KUKA KRL data list: ps_geo_c1.dat

&ACCESS RVO1
&REL 131
&COMMENT Solda GUN C1 geometria
&PARAM DISKPATH = KRC:\R1\Program
DEFDAT  ps_geo_c1
;FOLD EXTERNAL DECLARATIONS;%{PE}%MKUKATPBASIS,%CEXT,%VCOMMON,%P
;FOLD GRIPPERTECH EXT
EXT  H50 (INT  :IN,INT  :IN,INT  :IN,GRP_TYP  :IN )
;ENDFOLD (GRIPPERTECH EXT)
;FOLD SPOTTECH EXT
EXT  USERSPOT (S_COMMAND  :IN,SPOT_TYPE  :IN )
;ENDFOLD (SPOTTECH EXT)
;FOLD BASISTECH EXT;%{PE}%MKUKATPBASIS,%CEXT,%VEXT,%P
EXT  BAS (BAS_COMMAND  :IN,REAL  :IN )
DECL INT SUCCESS
;ENDFOLD (BASISTECH EXT)
;FOLD USER EXT;%{E}%MKUKATPUSER,%CEXT,%VEXT,%P
;Make your modifications here

;ENDFOLD (USER EXT)
;ENDFOLD (EXTERNAL DECLARATIONS)

;# ============ START PATH : swp_p13050r2_l_geo_c1 =============
DECL FDAT Fswp_60_5390={TOOL_NO 2,BASE_NO 1,IPO_FRAME #BASE,POINT2[] " ",TQ_STATE FALSE}
DECL SPOT_TYPE SS_OLP1={GUN 1,PAIR #FIRST,RETR #CLO,CLO_TM 0,PGNO1 1,PRESS1 1.0,PGNO2 0,PRESS2 0.0}
DECL E6POS Xswp_60_5390={X 1793.60498,Y 1119.29797,Z -41.4300003,A -165.905701,B -75.0368805,C 75.6208725,S 6,T 51,E1 -4282.88623,E2 0.0,E3 0.0,E4 0.0,E5 0.0,E6 0.0}
DECL FDAT Fswp_60_5378={TOOL_NO 2,BASE_NO 1,IPO_FRAME #BASE,POINT2[] " "}
DECL SPOT_TYPE SS_OLP2={GUN 1,PAIR #FIRST,RETR #CLO,CLO_TM 0,PGNO1 1,PRESS1 1.0,PGNO2 0,PRESS2 0.0}
DECL E6POS Xswp_60_5378={X 1995.44397,Y 1122.11902,Z -40.4609795,A -2.36140203,B -49.9265404,C -89.8133316,S 6,T 51,E1 -4282.31592,E2 0.0,E3 0.0,E4 0.0,E5 0.0,E6 0.0}
DECL FDAT Fswp_60_5368={TOOL_NO 2,BASE_NO 1,IPO_FRAME #BASE,POINT2[] " "}
DECL SPOT_TYPE SS_OLP3={GUN 1,PAIR #FIRST,RETR #CLO,CLO_TM 0,PGNO1 1,PRESS1 1.0,PGNO2 0,PRESS2 0.0}
DECL E6POS Xswp_60_5368={X 2052.64502,Y 972.549072,Z -42.4693718,A -85.639267,B -73.5025711,C -95.7587891,S 6,T 51,E1 -4487.2959,E2 0.0,E3 0.0,E4 0.0,E5 0.0,E6 0.0}
DECL FDAT Fswp_60_5360={TOOL_NO 2,BASE_NO 1,IPO_FRAME #BASE,POINT2[] " "}
DECL SPOT_TYPE SS_OLP4={GUN 1,PAIR #FIRST,RETR #CLO,CLO_TM 0,PGNO1 1,PRESS1 1.0,PGNO2 0,PRESS2 0.0}
DECL E6POS Xswp_60_5360={X 2051.40991,Y 830.991577,Z -72.7930908,A -89.8485336,B -38.7230415,C -92.0951614,S 6,T 51,E1 -4487.2959,E2 0.0,E3 0.0,E4 0.0,E5 0.0,E6 0.0}
DECL FDAT Fswp_60_5354={TOOL_NO 2,BASE_NO 1,IPO_FRAME #BASE,POINT2[] " "}
DECL SPOT_TYPE SS_OLP5={GUN 1,PAIR #FIRST,RETR #CLO,CLO_TM 0,PGNO1 1,PRESS1 1.0,PGNO2 0,PRESS2 0.0}
DECL E6POS Xswp_60_5354={X 2052.74707,Y 687.211487,Z -69.1016464,A 89.8141937,B -4.71356201,C 90.1745834,S 6,T 51,E1 -4487.2998,E2 0.0,E3 0.0,E4 0.0,E5 0.0,E6 0.0}
DECL FDAT Fswp_60_5348={TOOL_NO 2,BASE_NO 1,IPO_FRAME #BASE,POINT2[] " "}
DECL SPOT_TYPE SS_OLP6={GUN 1,PAIR #FIRST,RETR #CLO,CLO_TM 0,PGNO1 1,PRESS1 1.0,PGNO2 0,PRESS2 0.0}
DECL E6POS Xswp_60_5348={X 2051.51196,Y 627.115173,Z -2.50994706,A 89.8144608,B -4.71358299,C 90.1741791,S 6,T 51,E1 -4487.2998,E2 0.0,E3 0.0,E4 0.0,E5 0.0,E6 0.0}
DECL FDAT Fswp_60_5342={TOOL_NO 2,BASE_NO 1,IPO_FRAME #BASE,POINT2[] " "}
DECL SPOT_TYPE SS_OLP7={GUN 1,PAIR #FIRST,RETR #CLO,CLO_TM 0,PGNO1 1,PRESS1 1.0,PGNO2 0,PRESS2 0.0}
DECL E6POS Xswp_60_5342={X 2055.79199,Y 617.443176,Z 85.3936462,A 89.999321,B -34.127739,C 90.0019379,S 6,T 51,E1 -4487.30078,E2 0.0,E3 0.0,E4 0.0,E5 0.0,E6 0.0}
DECL FDAT Fswp_60_5336={TOOL_NO 2,BASE_NO 1,IPO_FRAME #BASE,POINT2[] " "}
DECL SPOT_TYPE SS_OLP8={GUN 1,PAIR #FIRST,RETR #CLO,CLO_TM 0,PGNO1 1,PRESS1 1.0,PGNO2 0,PRESS2 0.0}
DECL E6POS Xswp_60_5336={X 2058.30298,Y 508.353699,Z 145.004395,A 89.9974213,B -46.7444382,C 90.0027695,S 6,T 51,E1 -4487.2998,E2 0.0,E3 0.0,E4 0.0,E5 0.0,E6 0.0}
DECL SPOT_TYPE SS_OLP9={GUN 1,PAIR #FIRST,RETR #CLO,CLO_TM 0,PGNO1 1,PRESS1 1.0,PGNO2 0,PRESS2 0.0}
DECL FDAT Fswp_60_5324={TOOL_NO 2,BASE_NO 1,IPO_FRAME #BASE,POINT2[] " "}
DECL SPOT_TYPE SS_OLP10={GUN 1,PAIR #FIRST,RETR #CLO,CLO_TM 0,PGNO1 1,PRESS1 1.0,PGNO2 0,PRESS2 0.0}
DECL E6POS Xswp_60_5324={X 2058.63306,Y 416.970703,Z 279.76889,A 89.9949036,B -60.1505089,C 90.006073,S 6,T 51,E1 -4487.2998,E2 0.0,E3 0.0,E4 0.0,E5 0.0,E6 0.0}
DECL FDAT Fswp_60_5318={TOOL_NO 2,BASE_NO 1,IPO_FRAME #BASE,POINT2[] " "}
DECL SPOT_TYPE SS_OLP11={GUN 1,PAIR #FIRST,RETR #CLO,CLO_TM 0,PGNO1 1,PRESS1 1.0,PGNO2 0,PRESS2 0.0}
DECL E6POS Xswp_60_5318={X 2058.04297,Y 343.247498,Z 329.933685,A -89.9762192,B -84.4996567,C -90.0254974,S 6,T 51,E1 -4487.31787,E2 0.0,E3 0.0,E4 0.0,E5 0.0,E6 0.0}
DECL FDAT Fswp_60_5312={TOOL_NO 2,BASE_NO 1,IPO_FRAME #BASE,POINT2[] " "}
DECL SPOT_TYPE SS_OLP12={GUN 1,PAIR #FIRST,RETR #CLO,CLO_TM 0,PGNO1 1,PRESS1 1.0,PGNO2 0,PRESS2 0.0}
DECL E6POS Xswp_60_5312={X 2063.91699,Y 232.038406,Z 341.721008,A -90.0093765,B -89.2421036,C -89.9965515,S 6,T 51,E1 -4487.29785,E2 0.0,E3 0.0,E4 0.0,E5 0.0,E6 0.0}
DECL BASIS_SUGG_T LAST_BASIS={POINT1[] "P0                      ",POINT2[] "P0                      ",CP_PARAMS[] "CPDAT0                  ",PTP_PARAMS[] "PDAT0                   ",CONT[] "                        ",CP_VEL[] "2.0                     ",PTP_VEL[] "100                     ",SYNC_PARAMS[] "SYNCDAT                 ",SPL_NAME[] "S0                      "}
DECL SPOT_SUGG_T LAST_SPOT={GUN[] "1                       ",RETR_CMD[] "#OPN                    ",CHOISE[] "#FIRST                  ",CLO_TM[] "1                       ",PGNO1[] "37                      ",PRESS1[] "0                       ",PGNO2[] "1                       ",PRESS2[] "0                       ",SPOT_PARAMS[] "SDAT14                  "}
DECL SPOT_TYPE SSDAT1={GUN 1,PAIR #FIRST,RETR #OPN,CLO_TM 0,PGNO1 1,PRESS1 1.0,PGNO2 0,PRESS2 0.0}
DECL SPOT_TYPE SS_OLP13={GUN 1,PAIR #FIRST,RETR #CLO,CLO_TM 0,PGNO1 1,PRESS1 1.0,PGNO2 0,PRESS2 0.0}
DECL E6POS XP6={X 14.2474098,Y -4270.53809,Z 1356.71594,A 46.7418518,B 2.44693804,C -28.1381607,S 6,T 50,E1 -2092.58911,E2 0.0,E3 0.0,E4 0.0,E5 0.0,E6 0.0}
DECL FDAT FP6={TOOL_NO 2,BASE_NO 0,IPO_FRAME #BASE,POINT2[] " ",TQ_STATE FALSE}
DECL PDAT PPDAT34={VEL 100.0,ACC 100.0,APO_DIST 10.0,APO_MODE #CDIS}
DECL E6POS XPS123={X 1975.453,Y 1262.80505,Z -89.8548737,A -7.88512707,B -42.2266693,C -81.8771667,S 6,T 51,E1 -4282.896,E2 0.0,E3 0.0,E4 0.0,E5 0.0,E6 0.0}
DECL FDAT FPS123={TOOL_NO 2,BASE_NO 1,IPO_FRAME #BASE,POINT2[] " ",TQ_STATE FALSE}
DECL PDAT PPDAT38={VEL 100.0,ACC 100.0,APO_DIST 100.0}
DECL PDAT PPDAT0={VEL 100.0,ACC 100.0,APO_DIST 100.0,APO_MODE #CDIS}
DECL E6POS XP0={X 1831.76001,Y 1986.38696,Z 157.435593,A -57.9526711,B -77.0295563,C -42.9496689,S 6,T 50,E1 -4010.88403,E2 0.0,E3 0.0,E4 0.0,E5 0.0,E6 0.0}
DECL FDAT FP0={TOOL_NO 2,BASE_NO 1,IPO_FRAME #BASE,POINT2[] " ",TQ_STATE FALSE}
DECL E6POS XP10={X 1976.64001,Y 1119.03406,Z -90.3725662,A -5.75681591,B -42.5264511,C -84.9908371,S 6,T 51,E1 -4282.896,E2 0.0,E3 0.0,E4 0.0,E5 0.0,E6 0.0}
DECL FDAT FP10={TOOL_NO 2,BASE_NO 1,IPO_FRAME #BASE,POINT2[] " ",TQ_STATE FALSE}
DECL PDAT PPDAT39={VEL 100.0,ACC 100.0,APO_DIST 50.0,APO_MODE #CDIS}
DECL PDAT PPDAT40={VEL 100.0,ACC 100.0,APO_DIST 100.0}
DECL E6POS XP11={X 1931.23596,Y 1118.84595,Z -119.764801,A -12.6583996,B -41.2317009,C -74.8182831,S 6,T 51,E1 -4282.896,E2 0.0,E3 0.0,E4 0.0,E5 0.0,E6 0.0}
DECL FDAT FP11={TOOL_NO 2,BASE_NO 1,IPO_FRAME #BASE,POINT2[] " ",TQ_STATE FALSE}
DECL PDAT PPDAT41={VEL 100.0,ACC 100.0,APO_DIST 100.0,APO_MODE #CDIS}
DECL E6POS XP12={X 1819.70203,Y 1159.33301,Z -102.061302,A -82.8152771,B -72.2565918,C -9.40070915,S 6,T 51,E1 -4282.896,E2 0.0,E3 0.0,E4 0.0,E5 0.0,E6 0.0}
DECL FDAT FP12={TOOL_NO 2,BASE_NO 1,IPO_FRAME #BASE,POINT2[] " ",TQ_STATE FALSE}
DECL PDAT PPDAT42={VEL 100.0,ACC 100.0,APO_DIST 100.0,APO_MODE #CDIS}
DECL E6POS XP13={X 1792.13,Y 1120.06299,Z -64.8214035,A -155.350403,B -74.3082733,C 64.7092438,S 6,T 51,E1 -4282.896,E2 0.0,E3 0.0,E4 0.0,E5 0.0,E6 0.0}
DECL FDAT FP13={TOOL_NO 2,BASE_NO 1,IPO_FRAME #BASE,POINT2[] " ",TQ_STATE FALSE}
DECL PDAT PPDAT43={VEL 100.0,ACC 100.0,APO_DIST 100.0,APO_MODE #CDIS}
DECL PDAT PPDAT44={VEL 100.0,ACC 100.0,APO_DIST 100.0}
DECL E6POS XP14={X 1818.04395,Y 1135.521,Z -105.700798,A -167.004501,B -43.7118111,C 71.4859467,S 6,T 51,E1 -4282.896,E2 0.0,E3 0.0,E4 0.0,E5 0.0,E6 0.0}
DECL FDAT FP14={TOOL_NO 2,BASE_NO 1,IPO_FRAME #BASE,POINT2[] " ",TQ_STATE FALSE}
DECL PDAT PPDAT45={VEL 100.0,ACC 100.0,APO_DIST 100.0,APO_MODE #CDIS}
DECL E6POS XPS000={X 1814.72803,Y 1480.03296,Z -122.856003,A -167.018295,B -43.7061081,C 71.4881973,S 6,T 50,E1 -4282.896,E2 0.0,E3 0.0,E4 0.0,E5 0.0,E6 0.0}
DECL FDAT FPS000={TOOL_NO 2,BASE_NO 1,IPO_FRAME #BASE,POINT2[] " ",TQ_STATE FALSE}
DECL PDAT PPDAT46={VEL 100.0,ACC 100.0,APO_DIST 100.0}
DECL E6POS XP15={X 2255.78809,Y 2237.59106,Z 107.454803,A -82.0964432,B -22.1816597,C -22.13521,S 6,T 50,E1 -4282.89404,E2 0.0,E3 0.0,E4 0.0,E5 0.0,E6 0.0}
DECL FDAT FP15={TOOL_NO 2,BASE_NO 1,IPO_FRAME #BASE,POINT2[] " ",TQ_STATE FALSE}
DECL PDAT PPDAT47={VEL 100.0,ACC 100.0,APO_DIST 100.0,APO_MODE #CDIS}
DECL E6POS XP16={X 3165.62207,Y 1778.36902,Z -151.722107,A 120.920898,B -1.89024901,C 8.91728306,S 6,T 51,E1 -4282.89404,E2 0.0,E3 0.0,E4 0.0,E5 0.0,E6 0.0}
DECL FDAT FP16={TOOL_NO 2,BASE_NO 1,IPO_FRAME #BASE,POINT2[] " ",TQ_STATE FALSE}
DECL PDAT PPDAT49={VEL 100.0,ACC 100.0,APO_DIST 100.0,APO_MODE #CDIS}
DECL E6POS XP17={X 2850.94189,Y 1183.13403,Z -133.184601,A 127.037201,B -29.0648193,C 14.88025,S 6,T 51,E1 -4379.94092,E2 0.0,E3 0.0,E4 0.0,E5 0.0,E6 0.0}
DECL FDAT FP17={TOOL_NO 2,BASE_NO 1,IPO_FRAME #BASE,POINT2[] " ",TQ_STATE FALSE}
DECL PDAT PPDAT50={VEL 100.0,ACC 100.0,APO_DIST 100.0,APO_MODE #CDIS}
DECL E6POS XP18={X 2507.34912,Y 900.431274,Z -270.858887,A -154.130707,B -49.1211395,C -23.3417206,S 6,T 51,E1 -4427.95215,E2 0.0,E3 0.0,E4 0.0,E5 0.0,E6 0.0}
DECL FDAT FP18={TOOL_NO 2,BASE_NO 1,IPO_FRAME #BASE,POINT2[] " ",TQ_STATE FALSE}
DECL PDAT PPDAT51={VEL 100.0,ACC 100.0,APO_DIST 100.0,APO_MODE #CDIS}
DECL E6POS XP19={X 2244.12695,Y 845.446411,Z -102.626404,A -90.2177734,B -50.6062508,C -89.3426514,S 6,T 51,E1 -4487.2998,E2 0.0,E3 0.0,E4 0.0,E5 0.0,E6 0.0}
DECL FDAT FP19={TOOL_NO 2,BASE_NO 1,IPO_FRAME #BASE,POINT2[] " ",TQ_STATE FALSE}
DECL PDAT PPDAT52={VEL 100.0,ACC 100.0,APO_DIST 100.0,APO_MODE #CDIS}
DECL E6POS XP20={X 2115.19409,Y 940.910217,Z -73.8749466,A -88.6004715,B -57.4064102,C -93.0368729,S 6,T 51,E1 -4487.29688,E2 0.0,E3 0.0,E4 0.0,E5 0.0,E6 0.0}
DECL FDAT FP20={TOOL_NO 2,BASE_NO 1,IPO_FRAME #BASE,POINT2[] " ",TQ_STATE FALSE}
DECL PDAT PPDAT53={VEL 100.0,ACC 100.0,APO_DIST 100.0,APO_MODE #CDIS}
DECL E6POS XP21={X 2047.13098,Y 942.281982,Z -76.641983,A -88.6010895,B -57.405941,C -93.0353088,S 6,T 51,E1 -4487.29688,E2 0.0,E3 0.0,E4 0.0,E5 0.0,E6 0.0}
DECL FDAT FP21={TOOL_NO 2,BASE_NO 1,IPO_FRAME #BASE,POINT2[] " ",TQ_STATE FALSE}
DECL PDAT PPDAT54={VEL 100.0,ACC 100.0,APO_DIST 100.0,APO_MODE #CDIS}
DECL E6POS XP22={X 2047.75195,Y 982.460327,Z -49.2609482,A -85.6292114,B -73.5014267,C -95.7655716,S 6,T 51,E1 -4487.29688,E2 0.0,E3 0.0,E4 0.0,E5 0.0,E6 0.0}
DECL FDAT FP22={TOOL_NO 2,BASE_NO 1,IPO_FRAME #BASE,POINT2[] " ",TQ_STATE FALSE}
DECL PDAT PPDAT55={VEL 100.0,ACC 100.0,APO_DIST 100.0,APO_MODE #CDIS}
DECL PDAT PPDAT56={VEL 100.0,ACC 100.0,APO_DIST 100.0}
DECL E6POS XP23={X 2048.30591,Y 918.138916,Z -63.4876289,A -88.6876297,B -56.5051003,C -92.9628525,S 6,T 51,E1 -4487.29688,E2 0.0,E3 0.0,E4 0.0,E5 0.0,E6 0.0}
DECL FDAT FP23={TOOL_NO 2,BASE_NO 1,IPO_FRAME #BASE,POINT2[] " ",TQ_STATE FALSE}
DECL PDAT PPDAT57={VEL 100.0,ACC 100.0,APO_DIST 100.0,APO_MODE #CDIS}
DECL E6POS XP24={X 2049.125,Y 831.437378,Z -74.7315063,A -89.8483734,B -38.7232094,C -92.0950165,S 6,T 51,E1 -4487.29688,E2 0.0,E3 0.0,E4 0.0,E5 0.0,E6 0.0}
DECL FDAT FP24={TOOL_NO 2,BASE_NO 1,IPO_FRAME #BASE,POINT2[] " ",TQ_STATE FALSE}
DECL PDAT PPDAT58={VEL 100.0,ACC 100.0,APO_DIST 20.0,APO_MODE #CDIS}
DECL PDAT PPDAT59={VEL 100.0,ACC 100.0,APO_DIST 100.0}
DECL E6POS XP25={X 2046.797,Y 858.526917,Z -100.2687,A -89.9878235,B -36.5164413,C -90.7241592,S 6,T 51,E1 -4487.29883,E2 0.0,E3 0.0,E4 0.0,E5 0.0,E6 0.0}
DECL FDAT FP25={TOOL_NO 2,BASE_NO 1,IPO_FRAME #BASE,POINT2[] " ",TQ_STATE FALSE}
DECL PDAT PPDAT60={VEL 100.0,ACC 100.0,APO_DIST 100.0,APO_MODE #CDIS}
DECL E6POS XP26={X 2159.44507,Y 857.708984,Z -101.407303,A -89.9878235,B -36.5160408,C -90.7243576,S 6,T 51,E1 -4487.29883,E2 0.0,E3 0.0,E4 0.0,E5 0.0,E6 0.0}
DECL FDAT FP26={TOOL_NO 2,BASE_NO 1,IPO_FRAME #BASE,POINT2[] " ",TQ_STATE FALSE}
DECL PDAT PPDAT61={VEL 100.0,ACC 100.0,APO_DIST 100.0,APO_MODE #CDIS}
DECL E6POS XP27={X 2146.48999,Y 788.576416,Z -75.8830719,A 89.8144608,B -4.71849298,C 90.1741867,S 6,T 51,E1 -4487.2998,E2 0.0,E3 0.0,E4 0.0,E5 0.0,E6 0.0}
DECL FDAT FP27={TOOL_NO 2,BASE_NO 1,IPO_FRAME #BASE,POINT2[] " ",TQ_STATE FALSE}
DECL PDAT PPDAT62={VEL 100.0,ACC 100.0,APO_DIST 100.0,APO_MODE #CDIS}
DECL E6POS XP28={X 2146.62695,Y 811.116272,Z -52.6086311,A -88.3386993,B -84.5875397,C -91.8407135,S 6,T 51,E1 -4487.2998,E2 0.0,E3 0.0,E4 0.0,E5 0.0,E6 0.0}
DECL FDAT FP28={TOOL_NO 2,BASE_NO 1,IPO_FRAME #BASE,POINT2[] " ",TQ_STATE FALSE}
DECL PDAT PPDAT63={VEL 100.0,ACC 100.0,APO_DIST 100.0,APO_MODE #CDIS}
DECL E6POS XP34={X 2051.16992,Y 627.691772,Z -43.1946182,A 89.8142395,B -4.71378708,C 90.1743011,S 6,T 51,E1 -4487.2998,E2 0.0,E3 0.0,E4 0.0,E5 0.0,E6 0.0}
DECL FDAT FP34={TOOL_NO 2,BASE_NO 1,IPO_FRAME #BASE,POINT2[] " ",TQ_STATE FALSE}
DECL PDAT PPDAT65={VEL 100.0,ACC 100.0,APO_DIST 100.0,APO_MODE #CDIS}
DECL PDAT PPDAT66={VEL 100.0,ACC 100.0,APO_DIST 100.0}
DECL E6POS XP35={X 2053.42993,Y 537.918091,Z 14.90874,A 89.9957962,B -33.604599,C 90.0059662,S 6,T 51,E1 -4487.2998,E2 0.0,E3 0.0,E4 0.0,E5 0.0,E6 0.0}
DECL FDAT FP35={TOOL_NO 2,BASE_NO 1,IPO_FRAME #BASE,POINT2[] " ",TQ_STATE FALSE}
DECL PDAT PPDAT67={VEL 100.0,ACC 100.0,APO_DIST 100.0,APO_MODE #CDIS}
DECL PDAT PPDAT68={VEL 100.0,ACC 100.0,APO_DIST 100.0}
DECL PDAT PPDAT69={VEL 100.0,ACC 100.0,APO_DIST 100.0}
DECL PDAT PPDAT70={VEL 100.0,ACC 100.0,APO_DIST 100.0}
DECL E6POS Xswp_60_5350={X 2057.52295,Y 450.2948,Z 220.931,A 89.9962006,B -49.0321198,C 90.0046692,S 6,T 51,E1 -4487.2998,E2 0.0,E3 0.0,E4 0.0,E5 0.0,E6 0.0}
DECL FDAT Fswp_60_5350={TOOL_NO 2,BASE_NO 1,IPO_FRAME #BASE,POINT2[] " ",TQ_STATE FALSE}
DECL E6POS XP36={X 2056.47998,Y 464.042999,Z 176.894196,A 89.9945374,B -47.4184914,C 90.0042496,S 6,T 51,E1 -4487.2998,E2 0.0,E3 0.0,E4 0.0,E5 0.0,E6 0.0}
DECL FDAT FP36={TOOL_NO 2,BASE_NO 1,IPO_FRAME #BASE,POINT2[] " ",TQ_STATE FALSE}
DECL PDAT PPDAT71={VEL 100.0,ACC 100.0,APO_DIST 100.0,APO_MODE #CDIS}
DECL PDAT PPDAT72={VEL 100.0,ACC 100.0,APO_DIST 100.0}
DECL E6POS XP37={X 2058.99902,Y 355.600891,Z 263.370087,A -89.9917908,B -84.4970779,C -90.0120468,S 6,T 51,E1 -4487.2998,E2 0.0,E3 0.0,E4 0.0,E5 0.0,E6 0.0}
DECL FDAT FP37={TOOL_NO 2,BASE_NO 1,IPO_FRAME #BASE,POINT2[] " ",TQ_STATE FALSE}
DECL PDAT PPDAT73={VEL 100.0,ACC 100.0,APO_DIST 100.0,APO_MODE #CDIS}
DECL PDAT PPDAT74={VEL 100.0,ACC 100.0,APO_DIST 100.0}
DECL E6POS XP38={X 2061.27295,Y 355.603607,Z 263.36969,A -89.986618,B -84.4975433,C -90.0177231,S 6,T 51,E1 -4487.2998,E2 0.0,E3 0.0,E4 0.0,E5 0.0,E6 0.0}
DECL FDAT FP38={TOOL_NO 2,BASE_NO 1,IPO_FRAME #BASE,POINT2[] " ",TQ_STATE FALSE}
DECL PDAT PPDAT75={VEL 100.0,ACC 100.0,APO_DIST 100.0,APO_MODE #CDIS}
DECL E6POS XP39={X 2118.13599,Y 333.994293,Z 271.6651,A 89.993927,B -68.975502,C 89.9993362,S 6,T 51,E1 -4487.29883,E2 0.0,E3 0.0,E4 0.0,E5 0.0,E6 0.0}
DECL FDAT FP39={TOOL_NO 2,BASE_NO 1,IPO_FRAME #BASE,POINT2[] " ",TQ_STATE FALSE}
DECL PDAT PPDAT76={VEL 100.0,ACC 100.0,APO_DIST 100.0,APO_MODE #CDIS}
DECL E6POS XP40={X 2075.04004,Y 270.539215,Z 300.605988,A 89.9879303,B -79.5295181,C 90.0074005,S 6,T 51,E1 -4487.29688,E2 0.0,E3 0.0,E4 0.0,E5 0.0,E6 0.0}
DECL FDAT FP40={TOOL_NO 2,BASE_NO 1,IPO_FRAME #BASE,POINT2[] " ",TQ_STATE FALSE}
DECL PDAT PPDAT77={VEL 100.0,ACC 100.0,APO_DIST 100.0,APO_MODE #CDIS}
DECL E6POS XP41={X 2059.625,Y 272.974213,Z 316.043213,A 89.9944382,B -79.5298462,C 90.000267,S 6,T 51,E1 -4487.29688,E2 0.0,E3 0.0,E4 0.0,E5 0.0,E6 0.0}
DECL FDAT FP41={TOOL_NO 2,BASE_NO 1,IPO_FRAME #BASE,POINT2[] " ",TQ_STATE FALSE}
DECL PDAT PPDAT78={VEL 100.0,ACC 100.0,APO_DIST 100.0,APO_MODE #CDIS}
DECL PDAT PPDAT79={VEL 100.0,ACC 100.0,APO_DIST 100.0}
DECL E6POS XP42={X 2063.51611,Y -5007.45508,Z 639.768799,A -73.1590881,B -24.9932995,C -19.3749294,S 6,T 51,E1 -4487.2998,E2 0.0,E3 0.0,E4 0.0,E5 0.0,E6 0.0}
DECL FDAT FP42={TOOL_NO 2,BASE_NO 0,IPO_FRAME #BASE,POINT2[] " ",TQ_STATE FALSE}
DECL PDAT PPDAT80={VEL 100.0,ACC 100.0,APO_DIST 100.0,APO_MODE #CDIS}
DECL E6POS XP43={X 2507.71899,Y -6022.83203,Z 1824.85803,A -15.74121,B -87.3473587,C -74.6977615,S 6,T 51,E1 -4487.29785,E2 0.0,E3 0.0,E4 0.0,E5 0.0,E6 0.0}
DECL FDAT FP43={TOOL_NO 2,BASE_NO 0,IPO_FRAME #BASE,POINT2[] " ",TQ_STATE FALSE}
DECL PDAT PPDAT81={VEL 100.0,ACC 100.0,APO_DIST 100.0,APO_MODE #CDIS}
DECL E6POS XP44={X 3580.86401,Y 1344.72595,Z -359.380798,A -178.304504,B 6.4053278,C -5.48929977,S 6,T 51,E1 -4064.18311,E2 0.0,E3 0.0,E4 0.0,E5 0.0,E6 0.0}
DECL FDAT FP44={TOOL_NO 2,BASE_NO 1,IPO_FRAME #BASE,POINT2[] " ",TQ_STATE FALSE}
DECL PDAT PPDAT82={VEL 100.0,ACC 100.0,APO_DIST 100.0,APO_MODE #CDIS}
DECL E6POS XP45={X 3286.89404,Y 2001.38904,Z -150.2827,A 163.915298,B -15.1394901,C 24.9498901,S 6,T 51,E1 -3093.53003,E2 0.0,E3 0.0,E4 0.0,E5 0.0,E6 0.0}
DECL FDAT FP45={TOOL_NO 2,BASE_NO 1,IPO_FRAME #BASE,POINT2[] " ",TQ_STATE FALSE}
DECL PDAT PPDAT83={VEL 100.0,ACC 100.0,APO_DIST 100.0,APO_MODE #CDIS}
DECL E6POS XP46={X -97.4183807,Y -1779.59204,Z 959.895325,A -87.2605209,B -4.11820889,C -0.3932679,S 2,T 10,E1 -303.91449,E2 0.0,E3 0.0,E4 0.0,E5 0.0,E6 0.0}
DECL FDAT FP46={TOOL_NO 2,BASE_NO 0,IPO_FRAME #BASE,POINT2[] " ",TQ_STATE FALSE}
DECL PDAT PPDAT84={VEL 100.0,ACC 100.0,APO_DIST 100.0}
DECL PDAT PPDAT86={VEL 100.0,ACC 100.0,APO_DIST 100.0,APO_MODE #CDIS}
DECL E6POS XP48={X -353.518188,Y -4054.72705,Z 1005.86902,A -168.852097,B -23.8397598,C 40.0236511,S 2,T 2,E1 -1997.07104,E2 0.0,E3 0.0,E4 0.0,E5 0.0,E6 0.0}
DECL FDAT FP48={TOOL_NO 2,BASE_NO 0,IPO_FRAME #BASE,POINT2[] " ",TQ_STATE FALSE}
DECL PDAT PPDAT87={VEL 100.0,ACC 100.0,APO_DIST 100.0}
DECL E6POS XP49={X 2050.37793,Y 688.451599,Z -119.098396,A 89.8146667,B -4.71360588,C 90.1747589,S 6,T 51,E1 -4487.29883,E2 0.0,E3 0.0,E4 0.0,E5 0.0,E6 0.0}
DECL FDAT FP49={TOOL_NO 2,BASE_NO 1,IPO_FRAME #BASE,POINT2[] " ",TQ_STATE FALSE}
DECL PDAT PPDAT88={VEL 100.0,ACC 100.0,APO_DIST 100.0,APO_MODE #CDIS}
DECL E6POS XP51={X 2332.18311,Y 353.697693,Z -173.253296,A -156.103607,B -66.3182678,C -25.5800705,S 6,T 51,E1 -4487.29883,E2 0.0,E3 0.0,E4 0.0,E5 0.0,E6 0.0}
DECL FDAT FP51={TOOL_NO 2,BASE_NO 1,IPO_FRAME #BASE,POINT2[] " ",TQ_STATE FALSE}
DECL PDAT PPDAT90={VEL 100.0,ACC 100.0,APO_DIST 100.0}
ENDDAT
